FUNCTION Convert_BYTE_TO_REAL : BOOL
VAR_INPUT
	in : BYTE;
	out : REFERENCE TO REAL;
END_VAR
VAR
	converted : REAL;
END_VAR

converted := BYTE_TO_REAL(in);

IF (REAL_TO_BYTE(converted) <> in) THEN
	RETURN;
END_IF

out := converted;
Convert_BYTE_TO_REAL := TRUE;

END_FUNCTION

(* stored: Version 1.1.0.1, ProductVersion 3.1.4024.12
   POU Convert_BYTE_TO_REAL: Id {548371d1-bfde-4660-9ffc-be036b14e427}, SpecialFunc None *)
